FUNCTION_BLOCK EllipseFitting (* Composite FB wrapping other FBs *)
  (* Standard: 61499-2 *)
  (* Version 1.0, 2020-08-26, Administrator *)
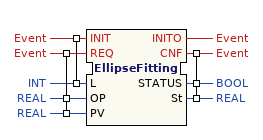
  EVENT_INPUT
    INIT WITH L; (* Initialization Request *)
    REQ WITH OP, PV; (* Normal Execution Request *)
  END_EVENT
  EVENT_OUTPUT
    INITO; (* Initialization Confirm *)
    CNF WITH STATUS, St; (* Execution Confirmation *)
  END_EVENT
  VAR_INPUT
    L : INT;
    OP : REAL; (* Input event qualifier *)
    PV : REAL;
  END_VAR
  VAR_OUTPUT
    STATUS : BOOL; (* Output event qualifier *)
    St : REAL;
  END_VAR
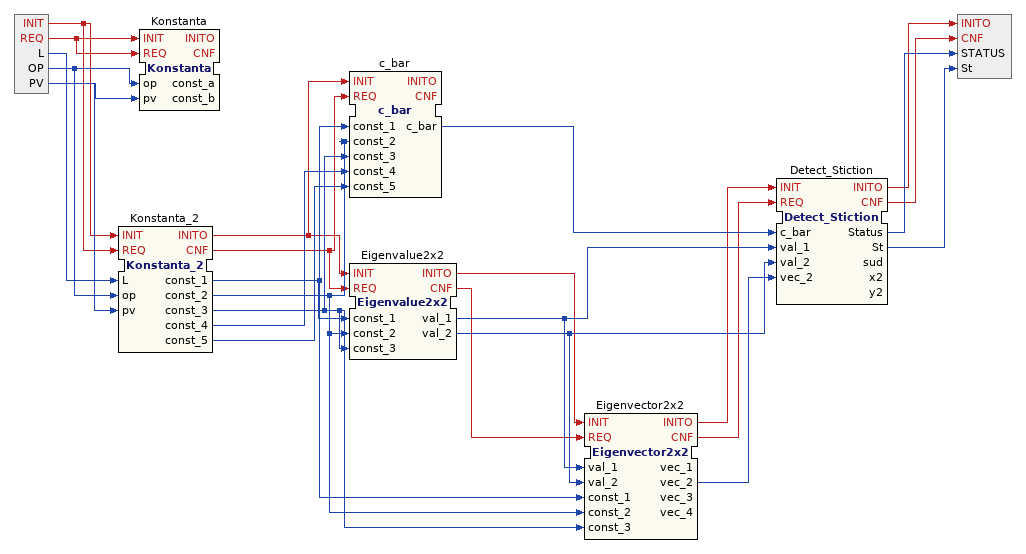
  FBS
    c_bar : c_bar;
    Eigenvalue2x2 : Eigenvalue2x2;
    Eigenvector2x2 : Eigenvector2x2;
    Konstanta : Konstanta;
    Konstanta_2 : Konstanta_2;
    Detect_Stiction : Detect_Stiction;
  END_FBS
  EVENT_CONNECTIONS
    Konstanta_2.CNF TO Eigenvalue2x2.REQ;
    Eigenvalue2x2.CNF TO Eigenvector2x2.REQ;
    Konstanta_2.INITO TO c_bar.INIT;
    Eigenvector2x2.INITO TO Detect_Stiction.INIT;
    Konstanta_2.INITO TO Eigenvalue2x2.INIT;
    Eigenvalue2x2.INITO TO Eigenvector2x2.INIT;
    Eigenvector2x2.CNF TO Detect_Stiction.REQ;
    Konstanta_2.CNF TO c_bar.REQ;
    Detect_Stiction.INITO TO INITO;
    Detect_Stiction.CNF TO CNF;
    REQ TO Konstanta_2.REQ;
    INIT TO Konstanta_2.INIT;
    REQ TO Konstanta.REQ;
    INIT TO Konstanta.INIT;
  END_CONNECTIONS
  DATA_CONNECTIONS
    Konstanta_2.const_3 TO c_bar.const_3;
    Konstanta_2.const_1 TO c_bar.const_1;
    Konstanta_2.const_3 TO Eigenvector2x2.const_3;
    Konstanta_2.const_2 TO Eigenvalue2x2.const_2;
    Konstanta_2.const_3 TO Eigenvalue2x2.const_3;
    Eigenvalue2x2.val_2 TO Eigenvector2x2.val_2;
    Eigenvalue2x2.val_1 TO Eigenvector2x2.val_1;
    Konstanta_2.const_2 TO Eigenvector2x2.const_2;
    c_bar.c_bar TO Detect_Stiction.c_bar;
    Konstanta_2.const_5 TO c_bar.const_5;
    Konstanta_2.const_4 TO c_bar.const_4;
    Konstanta_2.const_1 TO Eigenvalue2x2.const_1;
    Konstanta_2.const_1 TO Eigenvector2x2.const_1;
    Eigenvalue2x2.val_1 TO Detect_Stiction.val_1;
    Konstanta_2.const_2 TO c_bar.const_2;
    Eigenvector2x2.vec_2 TO Detect_Stiction.vec_2;
    Eigenvalue2x2.val_2 TO Detect_Stiction.val_2;
    L TO Konstanta_2.L;
    OP TO Konstanta_2.op;
    PV TO Konstanta_2.pv;
    OP TO Konstanta.op;
    PV TO Konstanta.pv;
    Detect_Stiction.Status TO STATUS;
    Detect_Stiction.St TO St;
  END_CONNECTIONS
END_FUNCTION_BLOCK
